FUNCTION_BLOCK NCITable
VAR_INPUT
END_VAR
VAR_OUTPUT
END_VAR
VAR
	nciTable : ST_NciFeedGroupTable;
END_VAR

;

END_FUNCTION_BLOCK

(* stored: Version 1.1.0.1, ProductVersion 3.1.4018.5
   POU NCITable: Id {4a7feab4-ad5e-44ea-b084-0a84be7b3292}, SpecialFunc None *)
